// Mitsubishi GX Works2 project: PROJECT   PLC: Q03UDV

PROGRAM MAIN
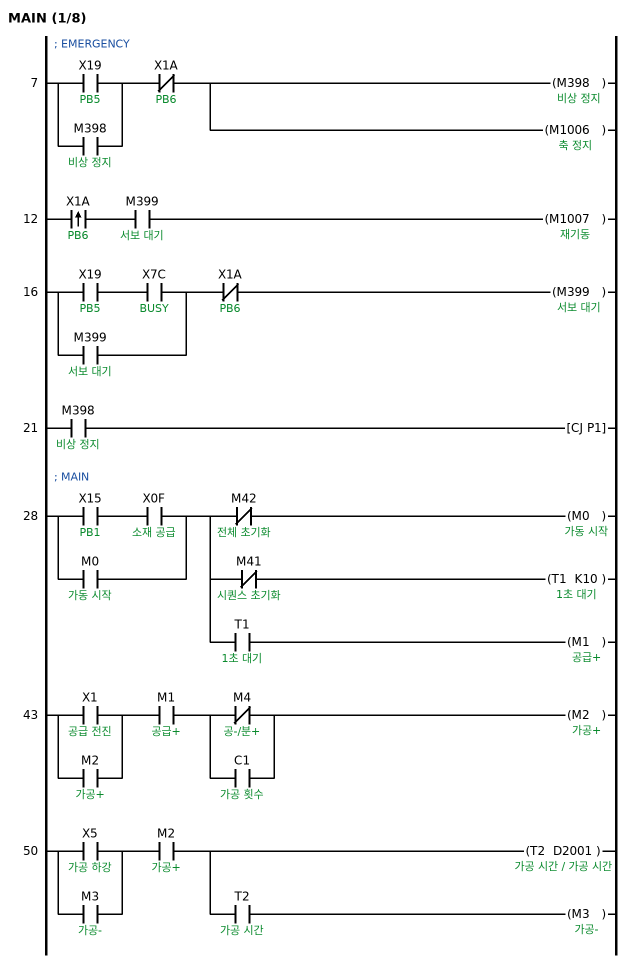
; EMERGENCY
7     LD      X19  ; PB5
      OR      M398  ; 비상 정지
      ANI     X1A  ; PB6
      OUT     M398  ; 비상 정지
      OUT     M1006  ; 축 정지
12    LDP     X1A  ; PB6
      AND     M399  ; 서보 대기
      OUT     M1007  ; 재기동
16    LD      X19  ; PB5
      AND     X7C  ; BUSY
      OR      M399  ; 서보 대기
      ANI     X1A  ; PB6
      OUT     M399  ; 서보 대기
21    LD      M398  ; 비상 정지
      CJ      P1  ; 비상 정지
; MAIN
28    LD      X15  ; PB1
      AND     X0F  ; 소재 공급
      OR      M0  ; 가동 시작
      MPS
      ANI     M42  ; 전체 초기화
      OUT     M0  ; 가동 시작
      MRD
      ANI     M41  ; 시퀀스 초기화
      OUT     T1 K10  ; 1초 대기
      MPP
      AND     T1  ; 1초 대기
      OUT     M1  ; 공급+
43    LD      X1  ; 공급 전진
      OR      M2  ; 가공+
      AND     M1  ; 공급+
      LDI     M4  ; 공-/분+
      OR      C1  ; 가공 횟수
      ANB
      OUT     M2  ; 가공+
50    LD      X5  ; 가공 하강
      OR      M3  ; 가공-
      AND     M2  ; 가공+
      OUT     T2 D2001  ; 가공 시간 / 가공 시간
      AND     T2  ; 가공 시간
      OUT     M3  ; 가공-
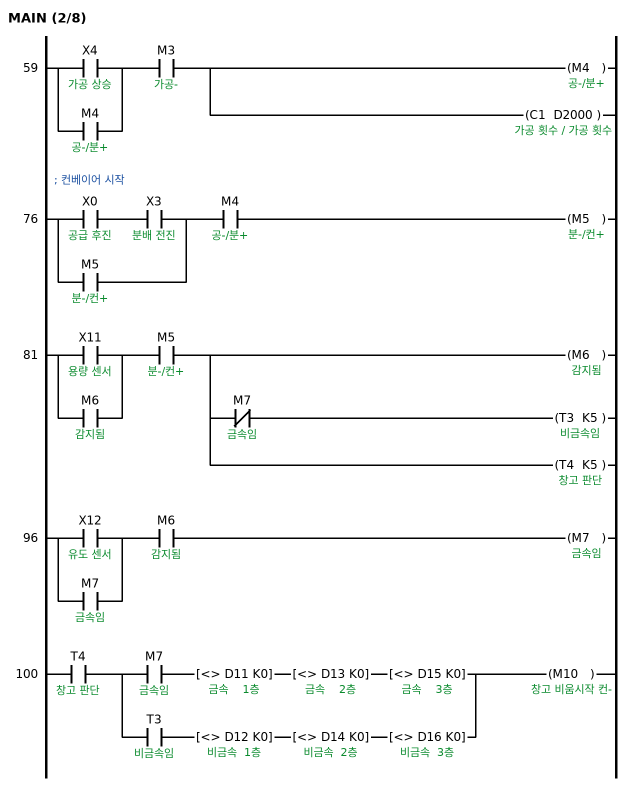
59    LD      X4  ; 가공 상승
      OR      M4  ; 공-/분+
      AND     M3  ; 가공-
      OUT     M4  ; 공-/분+
      OUT     C1 D2000  ; 가공 횟수 / 가공 횟수
; 컨베이어 시작
76    LD      X0  ; 공급 후진
      AND     X3  ; 분배 전진
      OR      M5  ; 분-/컨+
      AND     M4  ; 공-/분+
      OUT     M5  ; 분-/컨+
81    LD      X11  ; 용량 센서
      OR      M6  ; 감지됨
      AND     M5  ; 분-/컨+
      OUT     M6  ; 감지됨
      MPS
      ANI     M7  ; 금속임
      OUT     T3 K5  ; 비금속임
      MPP
      OUT     T4 K5  ; 창고 판단
96    LD      X12  ; 유도 센서
      OR      M7  ; 금속임
      AND     M6  ; 감지됨
      OUT     M7  ; 금속임
100   LD      T4  ; 창고 판단
      LD      M7  ; 금속임
      AND<>   D11 K0  ; 금속    1층
      AND<>   D13 K0  ; 금속    2층
      AND<>   D15 K0  ; 금속    3층
      LD      T3  ; 비금속임
      AND<>   D12 K0  ; 비금속  1층
      AND<>   D14 K0  ; 비금속  2층
      AND<>   D16 K0  ; 비금속  3층
      ORB
      ANB
      OUT     M10  ; 창고 비움시작 컨-
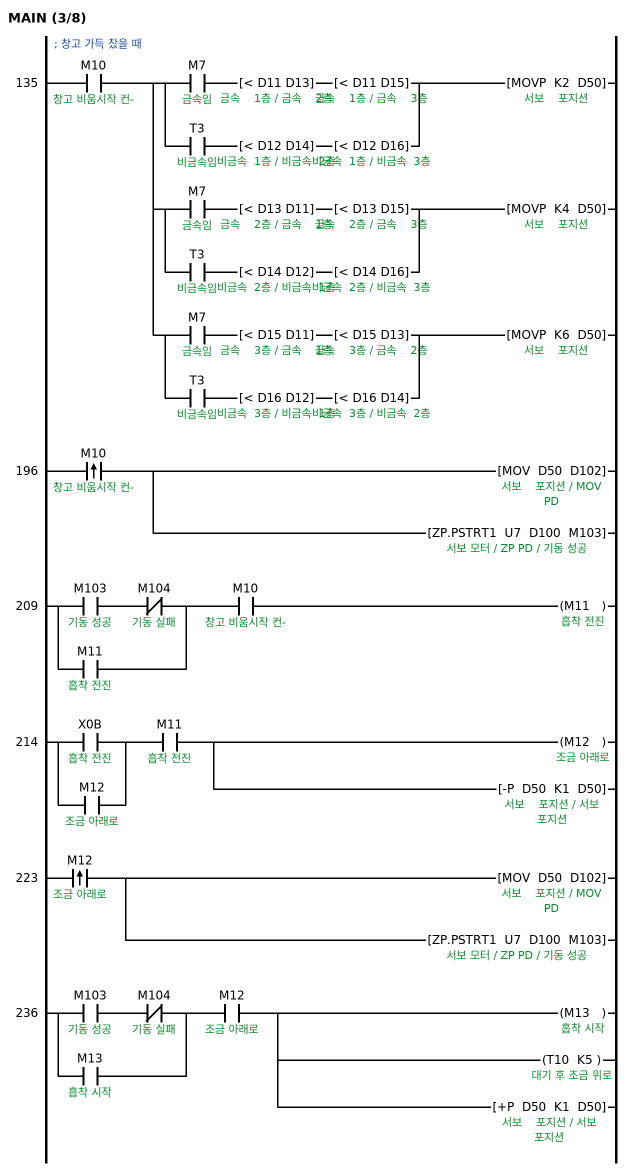
; 창고 가득 찼을 때
135   LD      M10  ; 창고 비움시작 컨-
      MPS
      LD      M7  ; 금속임
      AND<    D11 D13  ; 금속    1층 / 금속    2층
      AND<    D11 D15  ; 금속    1층 / 금속    3층
      LD      T3  ; 비금속임
      AND<    D12 D14  ; 비금속  1층 / 비금속  2층
      AND<    D12 D16  ; 비금속  1층 / 비금속  3층
      ORB
      ANB
      MOVP    K2 D50  ; 서보    포지션
      MRD
      LD      M7  ; 금속임
      AND<    D13 D11  ; 금속    2층 / 금속    1층
      AND<    D13 D15  ; 금속    2층 / 금속    3층
      LD      T3  ; 비금속임
      AND<    D14 D12  ; 비금속  2층 / 비금속  1층
      AND<    D14 D16  ; 비금속  2층 / 비금속  3층
      ORB
      ANB
      MOVP    K4 D50
      MPP
      LD      M7  ; 금속임
      AND<    D15 D11  ; 금속    3층 / 금속    1층
      AND<    D15 D13  ; 금속    3층 / 금속    2층
      LD      T3  ; 비금속임
      AND<    D16 D12  ; 비금속  3층 / 비금속  1층
      AND<    D16 D14  ; 비금속  3층 / 비금속  2층
      ORB
      ANB
      MOVP    K6 D50
196   LDP     M10  ; 창고 비움시작 컨-
      MOV     D50 D102  ; MOV PD
      ZP.PSTRT1 U7 D100 M103  ; 서보 모터 / ZP PD / 기동 성공
209   LD      M103  ; 기동 성공
      ANI     M104  ; 기동 실패
      OR      M11  ; 흡착 전진
      AND     M10  ; 창고 비움시작 컨-
      OUT     M11  ; 흡착 전진
214   LD      X0B  ; 흡착 전진
      OR      M12  ; 조금 아래로
      AND     M11  ; 흡착 전진
      OUT     M12  ; 조금 아래로
      -P      D50 K1 D50
223   LDP     M12  ; 조금 아래로
      MOV     D50 D102
      ZP.PSTRT1 U7 D100 M103
236   LD      M103  ; 기동 성공
      ANI     M104  ; 기동 실패
      OR      M13  ; 흡착 시작
      AND     M12  ; 조금 아래로
      OUT     M13  ; 흡착 시작
      OUT     T10 K5  ; 대기 후 조금 위로
      +P      D50 K1 D50
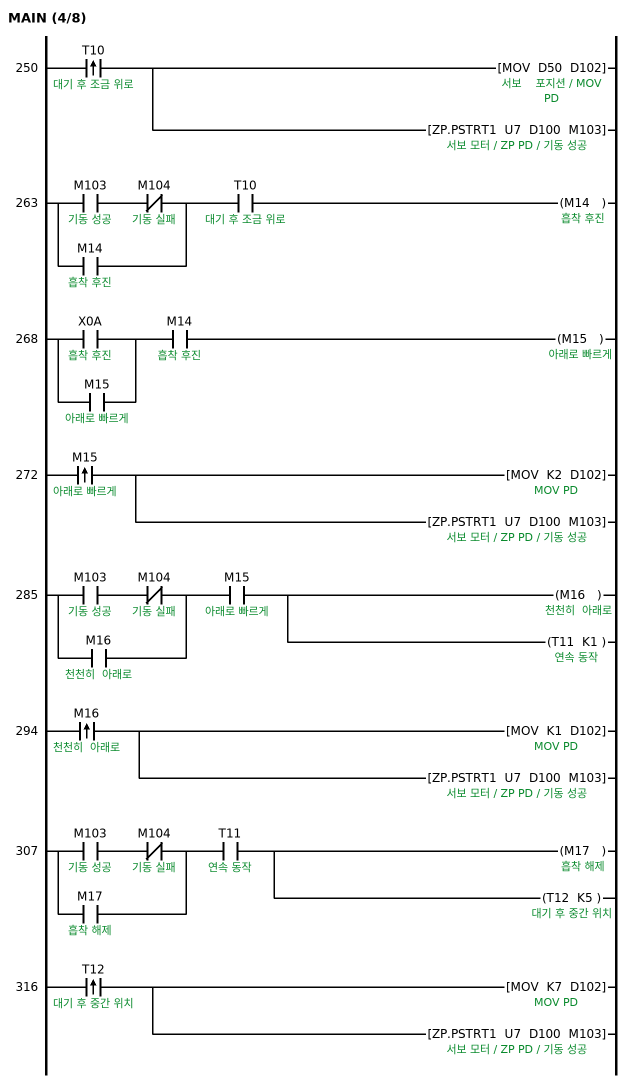
250   LDP     T10  ; 대기 후 조금 위로
      MOV     D50 D102
      ZP.PSTRT1 U7 D100 M103
263   LD      M103  ; 기동 성공
      ANI     M104  ; 기동 실패
      OR      M14  ; 흡착 후진
      AND     T10  ; 대기 후 조금 위로
      OUT     M14  ; 흡착 후진
268   LD      X0A  ; 흡착 후진
      OR      M15  ; 아래로 빠르게
      AND     M14  ; 흡착 후진
      OUT     M15  ; 아래로 빠르게
272   LDP     M15  ; 아래로 빠르게
      MOV     K2 D102
      ZP.PSTRT1 U7 D100 M103
285   LD      M103  ; 기동 성공
      ANI     M104  ; 기동 실패
      OR      M16  ; 천천히  아래로
      AND     M15  ; 아래로 빠르게
      OUT     M16  ; 천천히  아래로
      OUT     T11 K1  ; 연속 동작
294   LDP     M16  ; 천천히  아래로
      MOV     K1 D102
      ZP.PSTRT1 U7 D100 M103
307   LD      M103  ; 기동 성공
      ANI     M104  ; 기동 실패
      OR      M17  ; 흡착 해제
      AND     T11  ; 연속 동작
      OUT     M17  ; 흡착 해제
      OUT     T12 K5  ; 대기 후 중간 위치
316   LDP     T12  ; 대기 후 중간 위치
      MOV     K7 D102
      ZP.PSTRT1 U7 D100 M103
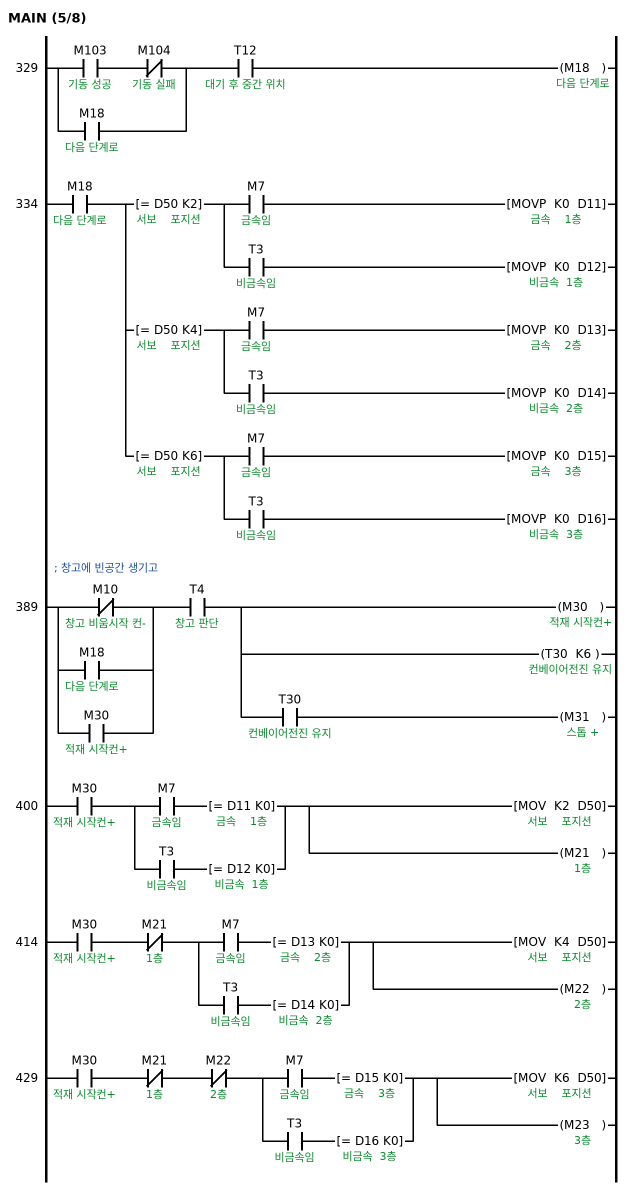
329   LD      M103  ; 기동 성공
      ANI     M104  ; 기동 실패
      OR      M18  ; 다음 단계로
      AND     T12  ; 대기 후 중간 위치
      OUT     M18  ; 다음 단계로
334   LD      M18  ; 다음 단계로
      MPS
      AND=    D50 K2  ; 서보    포지션
      MPS
      AND     M7  ; 금속임
      MOVP    K0 D11
      MPP
      AND     T3  ; 비금속임
      MOVP    K0 D12
      MRD
      AND=    D50 K4  ; 서보    포지션
      MPS
      AND     M7  ; 금속임
      MOVP    K0 D13
      MPP
      AND     T3  ; 비금속임
      MOVP    K0 D14
      MPP
      AND=    D50 K6  ; 서보    포지션
      MPS
      AND     M7  ; 금속임
      MOVP    K0 D15
      MPP
      AND     T3  ; 비금속임
      MOVP    K0 D16
; 창고에 빈공간 생기고
389   LDI     M10  ; 창고 비움시작 컨-
      OR      M18  ; 다음 단계로
      OR      M30  ; 적재 시작컨+
      AND     T4  ; 창고 판단
      OUT     M30  ; 적재 시작컨+
      OUT     T30 K6  ; 컨베이어전진 유지
      AND     T30  ; 컨베이어전진 유지
      OUT     M31  ; 스톱 +
400   LD      M30  ; 적재 시작컨+
      LD      M7  ; 금속임
      AND=    D11 K0  ; 금속    1층
      LD      T3  ; 비금속임
      AND=    D12 K0  ; 비금속  1층
      ORB
      ANB
      MOV     K2 D50
      OUT     M21  ; 1층
414   LD      M30  ; 적재 시작컨+
      ANI     M21  ; 1층
      LD      M7  ; 금속임
      AND=    D13 K0  ; 금속    2층
      LD      T3  ; 비금속임
      AND=    D14 K0  ; 비금속  2층
      ORB
      ANB
      MOV     K4 D50
      OUT     M22  ; 2층
429   LD      M30  ; 적재 시작컨+
      ANI     M21  ; 1층
      ANI     M22  ; 2층
      LD      M7  ; 금속임
      AND=    D15 K0  ; 금속    3층
      LD      T3  ; 비금속임
      AND=    D16 K0  ; 비금속  3층
      ORB
      ANB
      MOV     K6 D50
      OUT     M23  ; 3층
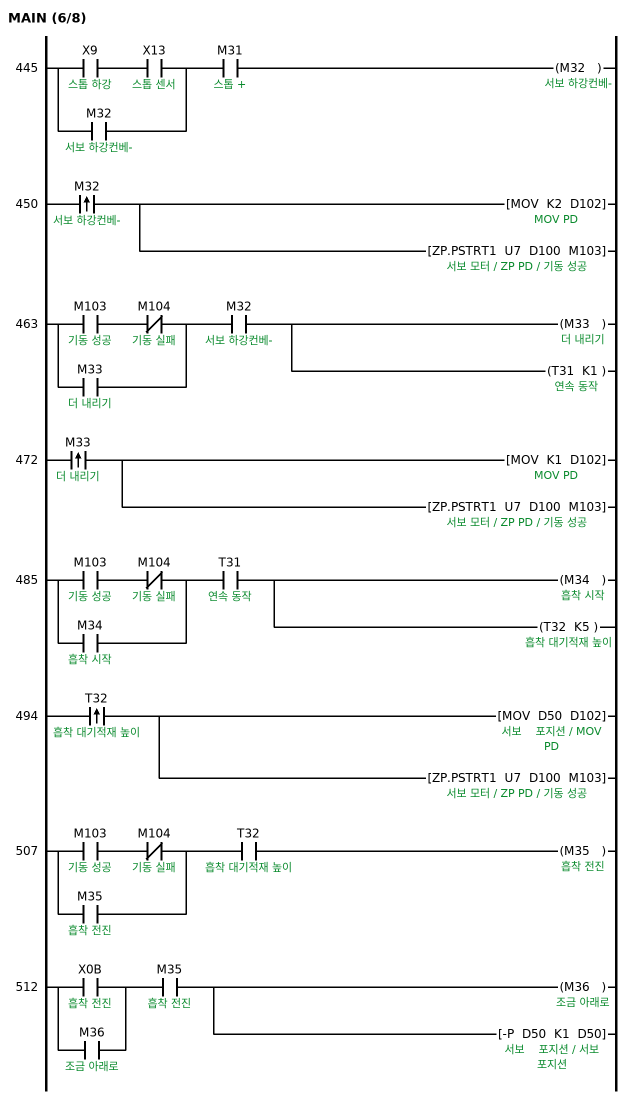
445   LD      X9  ; 스톱 하강
      AND     X13  ; 스톱 센서
      OR      M32  ; 서보 하강컨베-
      AND     M31  ; 스톱 +
      OUT     M32  ; 서보 하강컨베-
450   LDP     M32  ; 서보 하강컨베-
      MOV     K2 D102
      ZP.PSTRT1 U7 D100 M103
463   LD      M103  ; 기동 성공
      ANI     M104  ; 기동 실패
      OR      M33  ; 더 내리기
      AND     M32  ; 서보 하강컨베-
      OUT     M33  ; 더 내리기
      OUT     T31 K1  ; 연속 동작
472   LDP     M33  ; 더 내리기
      MOV     K1 D102
      ZP.PSTRT1 U7 D100 M103
485   LD      M103  ; 기동 성공
      ANI     M104  ; 기동 실패
      OR      M34  ; 흡착 시작
      AND     T31  ; 연속 동작
      OUT     M34  ; 흡착 시작
      OUT     T32 K5  ; 흡착 대기적재 높이
494   LDP     T32  ; 흡착 대기적재 높이
      MOV     D50 D102
      ZP.PSTRT1 U7 D100 M103
507   LD      M103  ; 기동 성공
      ANI     M104  ; 기동 실패
      OR      M35  ; 흡착 전진
      AND     T32  ; 흡착 대기적재 높이
      OUT     M35  ; 흡착 전진
512   LD      X0B  ; 흡착 전진
      OR      M36  ; 조금 아래로
      AND     M35  ; 흡착 전진
      OUT     M36  ; 조금 아래로
      -P      D50 K1 D50
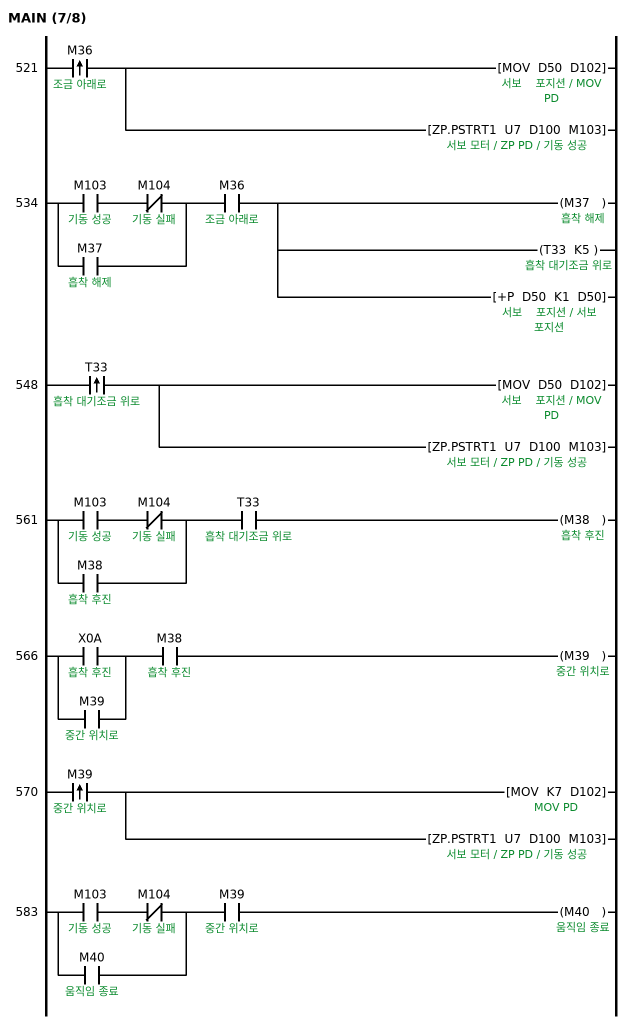
521   LDP     M36  ; 조금 아래로
      MOV     D50 D102
      ZP.PSTRT1 U7 D100 M103
534   LD      M103  ; 기동 성공
      ANI     M104  ; 기동 실패
      OR      M37  ; 흡착 해제
      AND     M36  ; 조금 아래로
      OUT     M37  ; 흡착 해제
      OUT     T33 K5  ; 흡착 대기조금 위로
      +P      D50 K1 D50
548   LDP     T33  ; 흡착 대기조금 위로
      MOV     D50 D102
      ZP.PSTRT1 U7 D100 M103
561   LD      M103  ; 기동 성공
      ANI     M104  ; 기동 실패
      OR      M38  ; 흡착 후진
      AND     T33  ; 흡착 대기조금 위로
      OUT     M38  ; 흡착 후진
566   LD      X0A  ; 흡착 후진
      OR      M39  ; 중간 위치로
      AND     M38  ; 흡착 후진
      OUT     M39  ; 중간 위치로
570   LDP     M39  ; 중간 위치로
      MOV     K7 D102
      ZP.PSTRT1 U7 D100 M103
583   LD      M103  ; 기동 성공
      ANI     M104  ; 기동 실패
      OR      M40  ; 움직임 종료
      AND     M39  ; 중간 위치로
      OUT     M40  ; 움직임 종료
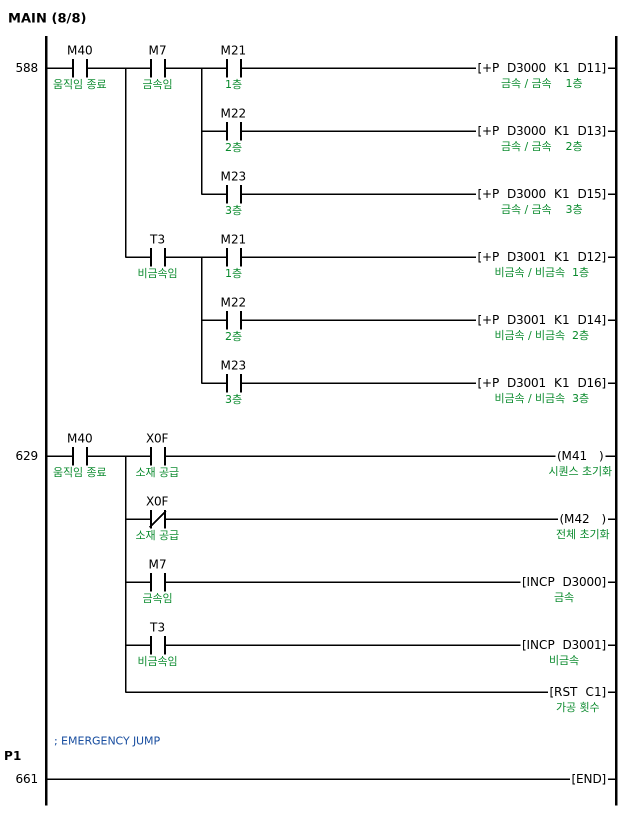
588   LD      M40  ; 움직임 종료
      MPS
      AND     M7  ; 금속임
      MPS
      AND     M21  ; 1층
      +P      D3000 K1 D11  ; 금속
      MRD
      AND     M22  ; 2층
      +P      D3000 K1 D13
      MPP
      AND     M23  ; 3층
      +P      D3000 K1 D15
      MPP
      AND     T3  ; 비금속임
      MPS
      AND     M21  ; 1층
      +P      D3001 K1 D12  ; 비금속
      MRD
      AND     M22  ; 2층
      +P      D3001 K1 D14
      MPP
      AND     M23  ; 3층
      +P      D3001 K1 D16
629   LD      M40  ; 움직임 종료
      MPS
      AND     X0F  ; 소재 공급
      OUT     M41  ; 시퀀스 초기화
      MRD
      ANI     X0F  ; 소재 공급
      OUT     M42  ; 전체 초기화
      MRD
      AND     M7  ; 금속임
      INCP    D3000
      MRD
      AND     T3  ; 비금속임
      INCP    D3001
      MPP
      RST     C1  ; 가공 횟수
; EMERGENCY JUMP
      P1
661   END
END_PROGRAM

PROGRAM INIT
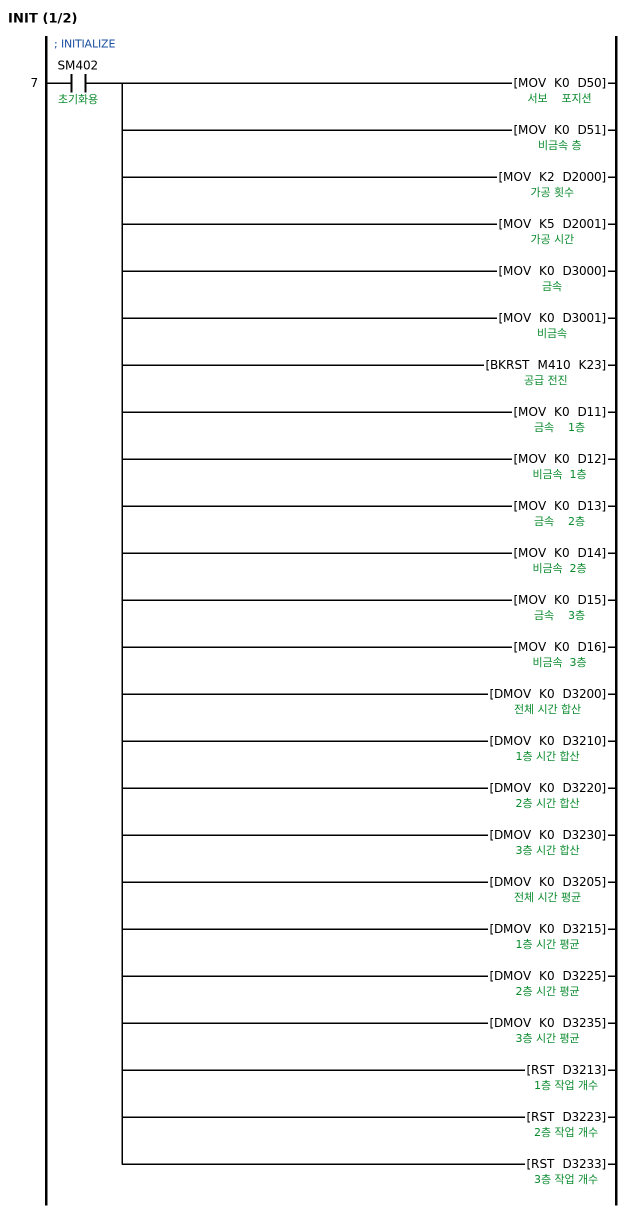
; INITIALIZE
7     LD      SM402  ; 초기화용
      MOV     K0 D50  ; 서보    포지션
      MOV     K0 D51  ; 비금속 층
      MOV     K2 D2000  ; 가공 횟수
      MOV     K5 D2001  ; 가공 시간
      MOV     K0 D3000  ; 금속
      MOV     K0 D3001  ; 비금속
      BKRST   M410 K23  ; 공급 전진
      MOV     K0 D11  ; 금속    1층
      MOV     K0 D12  ; 비금속  1층
      MOV     K0 D13  ; 금속    2층
      MOV     K0 D14  ; 비금속  2층
      MOV     K0 D15  ; 금속    3층
      MOV     K0 D16  ; 비금속  3층
      DMOV    K0 D3200  ; 전체 시간 합산
      DMOV    K0 D3210  ; 1층 시간 합산
      DMOV    K0 D3220  ; 2층 시간 합산
      DMOV    K0 D3230  ; 3층 시간 합산
      DMOV    K0 D3205  ; 전체 시간 평균
      DMOV    K0 D3215  ; 1층 시간 평균
      DMOV    K0 D3225  ; 2층 시간 평균
      DMOV    K0 D3235  ; 3층 시간 평균
      RST     D3213  ; 1층 작업 개수
      RST     D3223  ; 2층 작업 개수
      RST     D3233  ; 3층 작업 개수
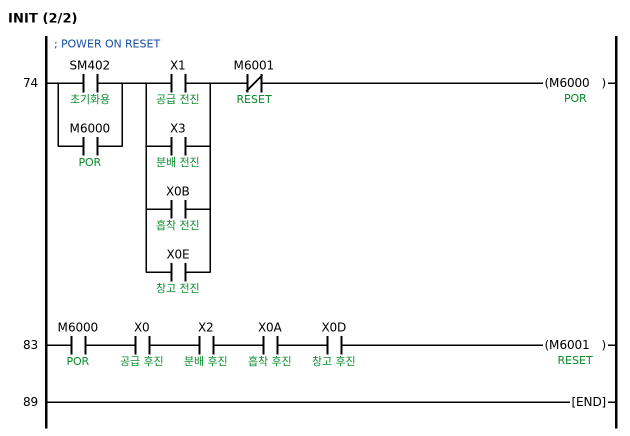
; POWER ON RESET
74    LD      SM402  ; 초기화용
      OR      M6000  ; POR
      LD      X1  ; 공급 전진
      OR      X3  ; 분배 전진
      OR      X0B  ; 흡착 전진
      OR      X0E  ; 창고 전진
      ANB
      ANI     M6001  ; RESET
      OUT     M6000  ; POR
83    LD      M6000  ; POR
      AND     X0  ; 공급 후진
      AND     X2  ; 분배 후진
      AND     X0A  ; 흡착 후진
      AND     X0D  ; 창고 후진
      OUT     M6001  ; RESET
89    END
END_PROGRAM

PROGRAM UNLOAD2
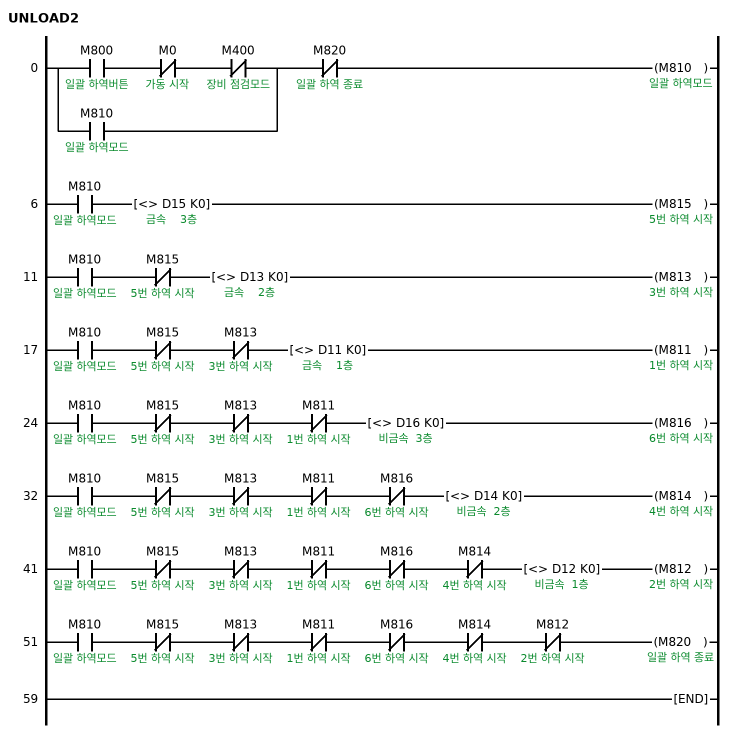
0     LD      M800  ; 일괄 하역버튼
      ANI     M0  ; 가동 시작
      ANI     M400  ; 장비 점검모드
      OR      M810  ; 일괄 하역모드
      ANI     M820  ; 일괄 하역 종료
      OUT     M810  ; 일괄 하역모드
6     LD      M810  ; 일괄 하역모드
      AND<>   D15 K0  ; 금속    3층
      OUT     M815  ; 5번 하역 시작
11    LD      M810  ; 일괄 하역모드
      ANI     M815  ; 5번 하역 시작
      AND<>   D13 K0  ; 금속    2층
      OUT     M813  ; 3번 하역 시작
17    LD      M810  ; 일괄 하역모드
      ANI     M815  ; 5번 하역 시작
      ANI     M813  ; 3번 하역 시작
      AND<>   D11 K0  ; 금속    1층
      OUT     M811  ; 1번 하역 시작
24    LD      M810  ; 일괄 하역모드
      ANI     M815  ; 5번 하역 시작
      ANI     M813  ; 3번 하역 시작
      ANI     M811  ; 1번 하역 시작
      AND<>   D16 K0  ; 비금속  3층
      OUT     M816  ; 6번 하역 시작
32    LD      M810  ; 일괄 하역모드
      ANI     M815  ; 5번 하역 시작
      ANI     M813  ; 3번 하역 시작
      ANI     M811  ; 1번 하역 시작
      ANI     M816  ; 6번 하역 시작
      AND<>   D14 K0  ; 비금속  2층
      OUT     M814  ; 4번 하역 시작
41    LD      M810  ; 일괄 하역모드
      ANI     M815  ; 5번 하역 시작
      ANI     M813  ; 3번 하역 시작
      ANI     M811  ; 1번 하역 시작
      ANI     M816  ; 6번 하역 시작
      ANI     M814  ; 4번 하역 시작
      AND<>   D12 K0  ; 비금속  1층
      OUT     M812  ; 2번 하역 시작
51    LD      M810  ; 일괄 하역모드
      ANI     M815  ; 5번 하역 시작
      ANI     M813  ; 3번 하역 시작
      ANI     M811  ; 1번 하역 시작
      ANI     M816  ; 6번 하역 시작
      ANI     M814  ; 4번 하역 시작
      ANI     M812  ; 2번 하역 시작
      OUT     M820  ; 일괄 하역 종료
59    END
END_PROGRAM

PROGRAM TEST
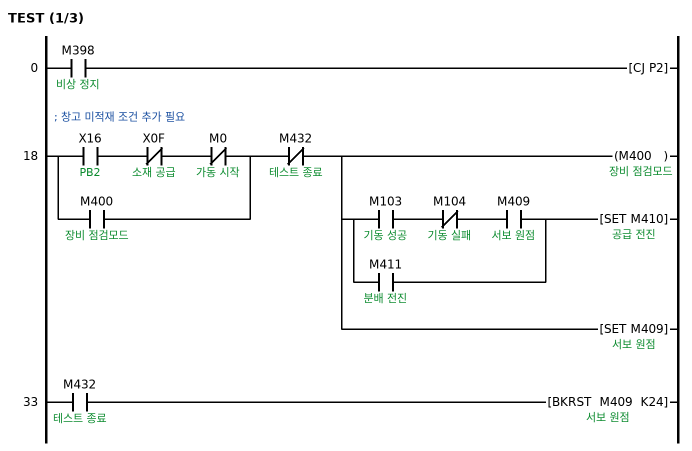
0     LD      M398  ; 비상 정지
      CJ      P2  ; 비상 정지
; 창고 미적재 조건 추가 필요
18    LD      X16  ; PB2
      ANI     X0F  ; 소재 공급
      ANI     M0  ; 가동 시작
      OR      M400  ; 장비 점검모드
      ANI     M432  ; 테스트 종료
      OUT     M400  ; 장비 점검모드
      MPS
      LD      M103  ; 기동 성공
      ANI     M104  ; 기동 실패
      AND     M409  ; 서보 원점
      OR      M411  ; 분배 전진
      ANB
      SET     M410  ; 공급 전진
      MPP
      SET     M409  ; 서보 원점
33    LD      M432  ; 테스트 종료
      BKRST   M409 K24
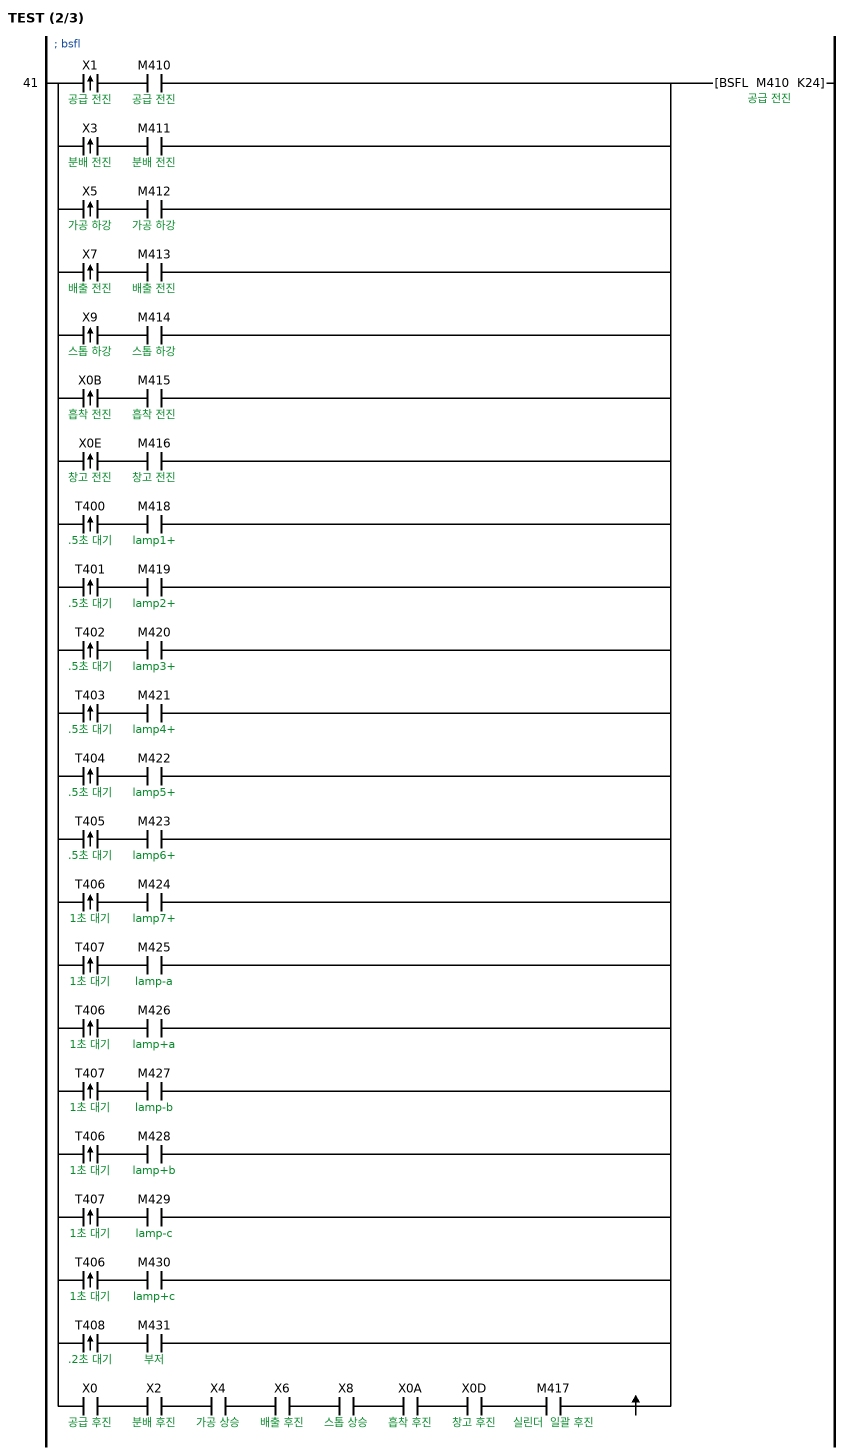
; bsfl
41    LDP     X1  ; 공급 전진
      AND     M410  ; 공급 전진
      LDP     X3  ; 분배 전진
      AND     M411  ; 분배 전진
      ORB
      LDP     X5  ; 가공 하강
      AND     M412  ; 가공 하강
      ORB
      LDP     X7  ; 배출 전진
      AND     M413  ; 배출 전진
      ORB
      LDP     X9  ; 스톱 하강
      AND     M414  ; 스톱 하강
      ORB
      LDP     X0B  ; 흡착 전진
      AND     M415  ; 흡착 전진
      ORB
      LDP     X0E  ; 창고 전진
      AND     M416  ; 창고 전진
      ORB
      LDP     T400  ; .5초 대기
      AND     M418  ; lamp1+
      ORB
      LDP     T401  ; .5초 대기
      AND     M419  ; lamp2+
      ORB
      LDP     T402  ; .5초 대기
      AND     M420  ; lamp3+
      ORB
      LDP     T403  ; .5초 대기
      AND     M421  ; lamp4+
      ORB
      LDP     T404  ; .5초 대기
      AND     M422  ; lamp5+
      ORB
      LDP     T405  ; .5초 대기
      AND     M423  ; lamp6+
      ORB
      LDP     T406  ; 1초 대기
      AND     M424  ; lamp7+
      ORB
      LDP     T407  ; 1초 대기
      AND     M425  ; lamp-a
      ORB
      LDP     T406  ; 1초 대기
      AND     M426  ; lamp+a
      ORB
      LDP     T407  ; 1초 대기
      AND     M427  ; lamp-b
      ORB
      LDP     T406  ; 1초 대기
      AND     M428  ; lamp+b
      ORB
      LDP     T407  ; 1초 대기
      AND     M429  ; lamp-c
      ORB
      LDP     T406  ; 1초 대기
      AND     M430  ; lamp+c
      ORB
      LDP     T408  ; .2초 대기
      AND     M431  ; 부저
      ORB
      LD      X0  ; 공급 후진
      AND     X2  ; 분배 후진
      AND     X4  ; 가공 상승
      AND     X6  ; 배출 후진
      AND     X8  ; 스톱 상승
      AND     X0A  ; 흡착 후진
      AND     X0D  ; 창고 후진
      AND     M417  ; 실린더  일괄 후진
      MEP
      ORB
      BSFL    M410 K24
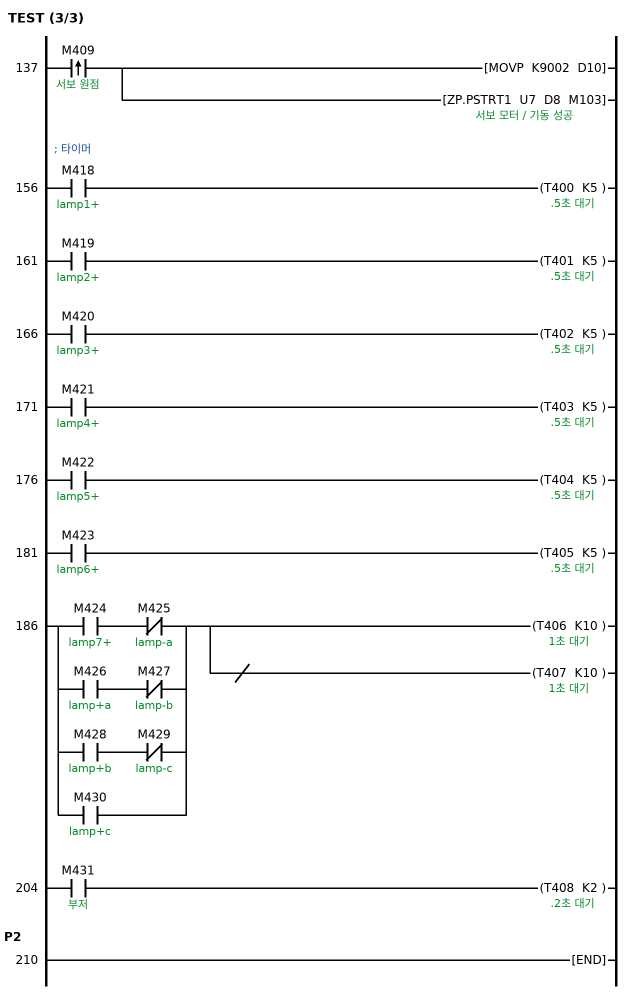
137   LDP     M409  ; 서보 원점
      MOVP    K9002 D10
      ZP.PSTRT1 U7 D8 M103  ; 서보 모터
; 타이머
156   LD      M418  ; lamp1+
      OUT     T400 K5  ; .5초 대기
161   LD      M419  ; lamp2+
      OUT     T401 K5  ; .5초 대기
166   LD      M420  ; lamp3+
      OUT     T402 K5  ; .5초 대기
171   LD      M421  ; lamp4+
      OUT     T403 K5  ; .5초 대기
176   LD      M422  ; lamp5+
      OUT     T404 K5  ; .5초 대기
181   LD      M423  ; lamp6+
      OUT     T405 K5  ; .5초 대기
186   LD      M424  ; lamp7+
      ANI     M425  ; lamp-a
      LD      M426  ; lamp+a
      ANI     M427  ; lamp-b
      ORB
      LD      M428  ; lamp+b
      ANI     M429  ; lamp-c
      ORB
      OR      M430  ; lamp+c
      OUT     T406 K10  ; 1초 대기
      INV
      OUT     T407 K10  ; 1초 대기
204   LD      M431  ; 부저
      OUT     T408 K2  ; .2초 대기
      P2
210   END
END_PROGRAM

PROGRAM OUTPUT
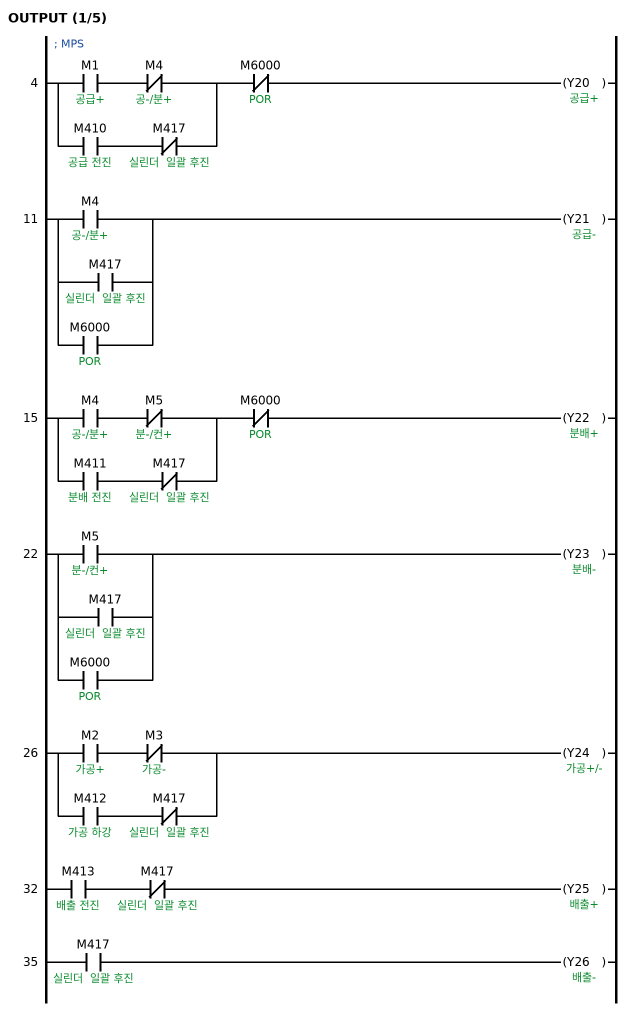
; MPS
4     LD      M1  ; 공급+
      ANI     M4  ; 공-/분+
      LD      M410  ; 공급 전진
      ANI     M417  ; 실린더  일괄 후진
      ORB
      ANI     M6000  ; POR
      OUT     Y20  ; 공급+
11    LD      M4  ; 공-/분+
      OR      M417  ; 실린더  일괄 후진
      OR      M6000  ; POR
      OUT     Y21  ; 공급-
15    LD      M4  ; 공-/분+
      ANI     M5  ; 분-/컨+
      LD      M411  ; 분배 전진
      ANI     M417  ; 실린더  일괄 후진
      ORB
      ANI     M6000  ; POR
      OUT     Y22  ; 분배+
22    LD      M5  ; 분-/컨+
      OR      M417  ; 실린더  일괄 후진
      OR      M6000  ; POR
      OUT     Y23  ; 분배-
26    LD      M2  ; 가공+
      ANI     M3  ; 가공-
      LD      M412  ; 가공 하강
      ANI     M417  ; 실린더  일괄 후진
      ORB
      OUT     Y24  ; 가공+/-
32    LD      M413  ; 배출 전진
      ANI     M417  ; 실린더  일괄 후진
      OUT     Y25  ; 배출+
35    LD      M417  ; 실린더  일괄 후진
      OUT     Y26  ; 배출-
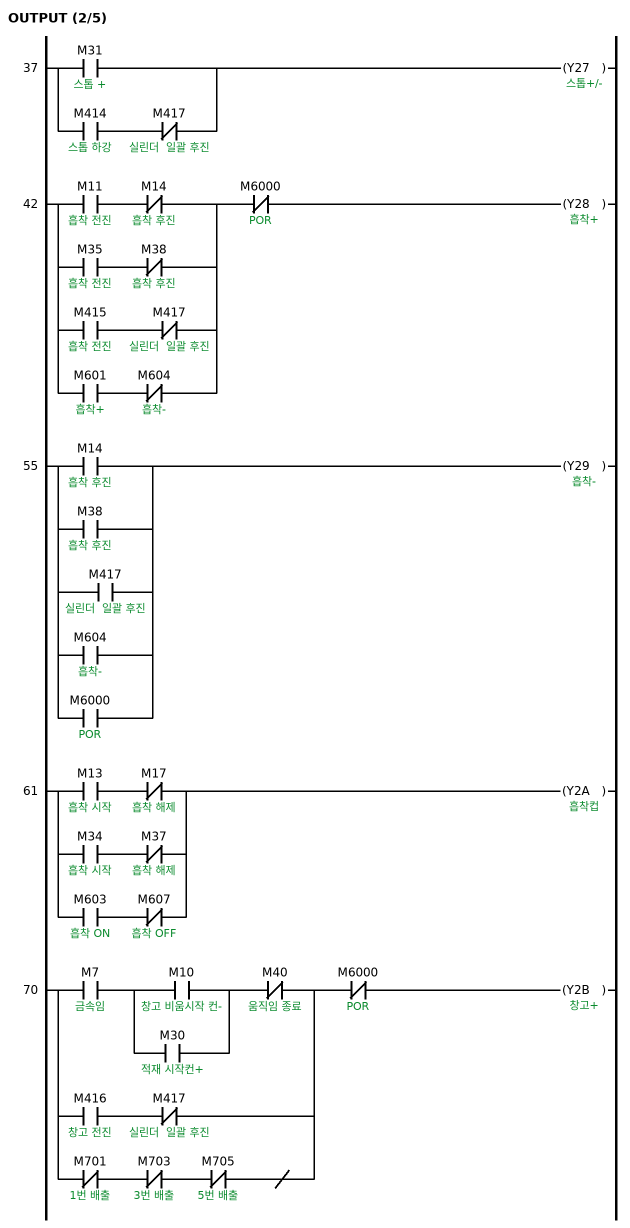
37    LD      M31  ; 스톱 +
      LD      M414  ; 스톱 하강
      ANI     M417  ; 실린더  일괄 후진
      ORB
      OUT     Y27  ; 스톱+/-
42    LD      M11  ; 흡착 전진
      ANI     M14  ; 흡착 후진
      LD      M35  ; 흡착 전진
      ANI     M38  ; 흡착 후진
      ORB
      LD      M415  ; 흡착 전진
      ANI     M417  ; 실린더  일괄 후진
      ORB
      LD      M601  ; 흡착+
      ANI     M604  ; 흡착-
      ORB
      ANI     M6000  ; POR
      OUT     Y28  ; 흡착+
55    LD      M14  ; 흡착 후진
      OR      M38  ; 흡착 후진
      OR      M417  ; 실린더  일괄 후진
      OR      M604  ; 흡착-
      OR      M6000  ; POR
      OUT     Y29  ; 흡착-
61    LD      M13  ; 흡착 시작
      ANI     M17  ; 흡착 해제
      LD      M34  ; 흡착 시작
      ANI     M37  ; 흡착 해제
      ORB
      LD      M603  ; 흡착 ON
      ANI     M607  ; 흡착 OFF
      ORB
      OUT     Y2A  ; 흡착컵
70    LD      M7  ; 금속임
      LD      M10  ; 창고 비움시작 컨-
      OR      M30  ; 적재 시작컨+
      ANB
      ANI     M40  ; 움직임 종료
      LD      M416  ; 창고 전진
      ANI     M417  ; 실린더  일괄 후진
      ORB
      LDI     M701  ; 1번 배출
      ANI     M703  ; 3번 배출
      ANI     M705  ; 5번 배출
      INV
      ORB
      ANI     M6000  ; POR
      OUT     Y2B  ; 창고+
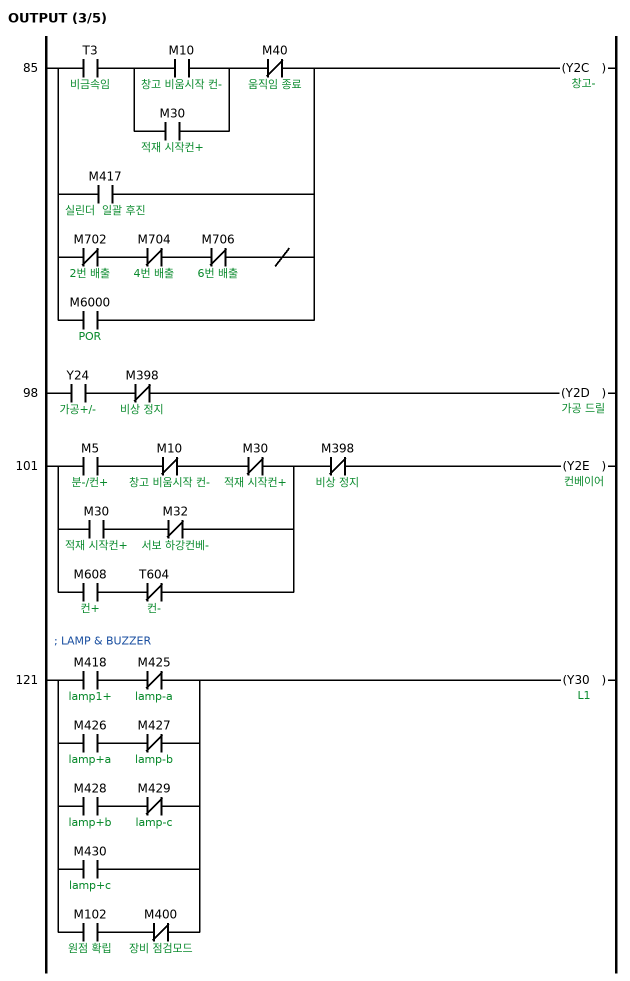
85    LD      T3  ; 비금속임
      LD      M10  ; 창고 비움시작 컨-
      OR      M30  ; 적재 시작컨+
      ANB
      ANI     M40  ; 움직임 종료
      OR      M417  ; 실린더  일괄 후진
      LDI     M702  ; 2번 배출
      ANI     M704  ; 4번 배출
      ANI     M706  ; 6번 배출
      INV
      ORB
      OR      M6000  ; POR
      OUT     Y2C  ; 창고-
98    LD      Y24  ; 가공+/-
      ANI     M398  ; 비상 정지
      OUT     Y2D  ; 가공 드릴
101   LD      M5  ; 분-/컨+
      ANI     M10  ; 창고 비움시작 컨-
      ANI     M30  ; 적재 시작컨+
      LD      M30  ; 적재 시작컨+
      ANI     M32  ; 서보 하강컨베-
      ORB
      LD      M608  ; 컨+
      ANI     T604  ; 컨-
      ORB
      ANI     M398  ; 비상 정지
      OUT     Y2E  ; 컨베이어
; LAMP & BUZZER
121   LD      M418  ; lamp1+
      ANI     M425  ; lamp-a
      LD      M426  ; lamp+a
      ANI     M427  ; lamp-b
      ORB
      LD      M428  ; lamp+b
      ANI     M429  ; lamp-c
      ORB
      OR      M430  ; lamp+c
      LD      M102  ; 원점 확립
      ANI     M400  ; 장비 점검모드
      ORB
      OUT     Y30  ; L1
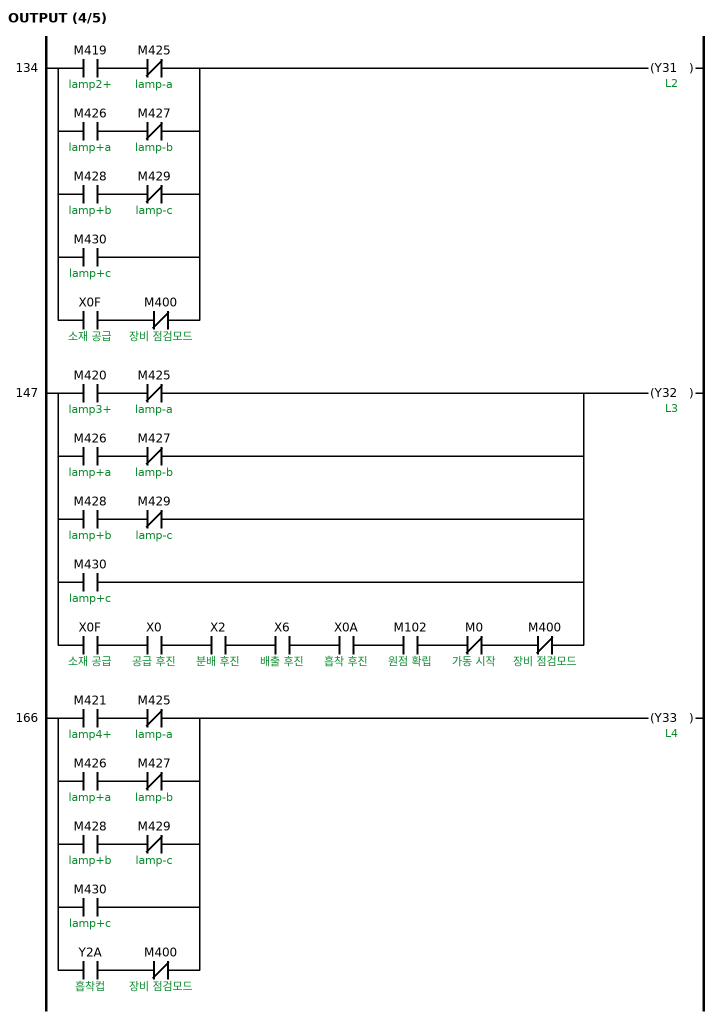
134   LD      M419  ; lamp2+
      ANI     M425  ; lamp-a
      LD      M426  ; lamp+a
      ANI     M427  ; lamp-b
      ORB
      LD      M428  ; lamp+b
      ANI     M429  ; lamp-c
      ORB
      OR      M430  ; lamp+c
      LD      X0F  ; 소재 공급
      ANI     M400  ; 장비 점검모드
      ORB
      OUT     Y31  ; L2
147   LD      M420  ; lamp3+
      ANI     M425  ; lamp-a
      LD      M426  ; lamp+a
      ANI     M427  ; lamp-b
      ORB
      LD      M428  ; lamp+b
      ANI     M429  ; lamp-c
      ORB
      OR      M430  ; lamp+c
      LD      X0F  ; 소재 공급
      AND     X0  ; 공급 후진
      AND     X2  ; 분배 후진
      AND     X6  ; 배출 후진
      AND     X0A  ; 흡착 후진
      AND     M102  ; 원점 확립
      ANI     M0  ; 가동 시작
      ANI     M400  ; 장비 점검모드
      ORB
      OUT     Y32  ; L3
166   LD      M421  ; lamp4+
      ANI     M425  ; lamp-a
      LD      M426  ; lamp+a
      ANI     M427  ; lamp-b
      ORB
      LD      M428  ; lamp+b
      ANI     M429  ; lamp-c
      ORB
      OR      M430  ; lamp+c
      LD      Y2A  ; 흡착컵
      ANI     M400  ; 장비 점검모드
      ORB
      OUT     Y33  ; L4
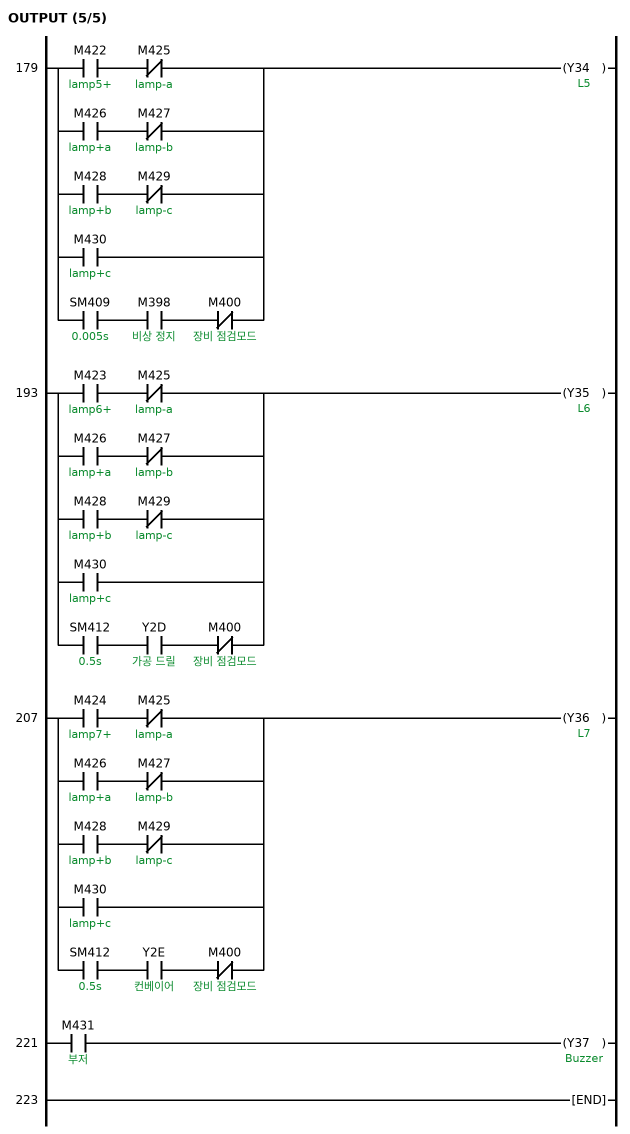
179   LD      M422  ; lamp5+
      ANI     M425  ; lamp-a
      LD      M426  ; lamp+a
      ANI     M427  ; lamp-b
      ORB
      LD      M428  ; lamp+b
      ANI     M429  ; lamp-c
      ORB
      OR      M430  ; lamp+c
      LD      SM409  ; 0.005s
      AND     M398  ; 비상 정지
      ANI     M400  ; 장비 점검모드
      ORB
      OUT     Y34  ; L5
193   LD      M423  ; lamp6+
      ANI     M425  ; lamp-a
      LD      M426  ; lamp+a
      ANI     M427  ; lamp-b
      ORB
      LD      M428  ; lamp+b
      ANI     M429  ; lamp-c
      ORB
      OR      M430  ; lamp+c
      LD      SM412  ; 0.5s
      AND     Y2D  ; 가공 드릴
      ANI     M400  ; 장비 점검모드
      ORB
      OUT     Y35  ; L6
207   LD      M424  ; lamp7+
      ANI     M425  ; lamp-a
      LD      M426  ; lamp+a
      ANI     M427  ; lamp-b
      ORB
      LD      M428  ; lamp+b
      ANI     M429  ; lamp-c
      ORB
      OR      M430  ; lamp+c
      LD      SM412  ; 0.5s
      AND     Y2E  ; 컨베이어
      ANI     M400  ; 장비 점검모드
      ORB
      OUT     Y36  ; L7
221   LD      M431  ; 부저
      OUT     Y37  ; Buzzer
223   END
END_PROGRAM

PROGRAM STAT
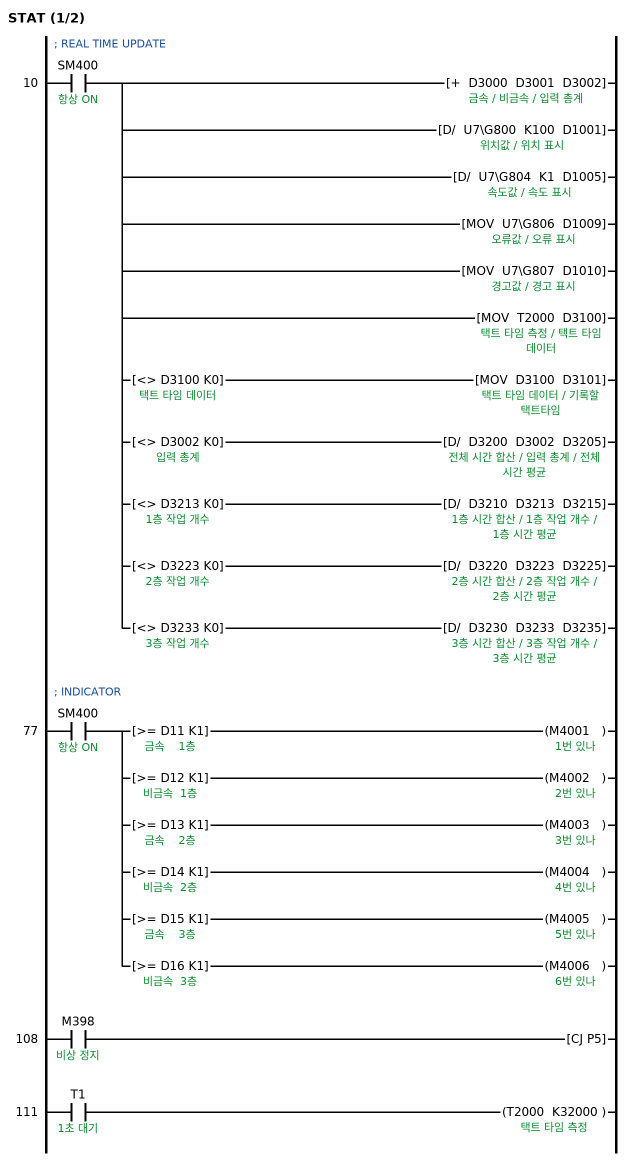
; REAL TIME UPDATE
10    LD      SM400  ; 항상 ON
      +       D3000 D3001 D3002  ; 금속 / 비금속 / 입력 총계
      D/      U7\G800 K100 D1001  ; 위치값 / 위치 표시
      D/      U7\G804 K1 D1005  ; 속도값 / 속도 표시
      MOV     U7\G806 D1009  ; 오류값 / 오류 표시
      MOV     U7\G807 D1010  ; 경고값 / 경고 표시
      MOV     T2000 D3100  ; 택트 타임 측정 / 택트 타임 데이터
      MPS
      AND<>   D3100 K0  ; 택트 타임 데이터
      MOV     D3100 D3101  ; 기록할  택트타임
      MRD
      AND<>   D3002 K0  ; 입력 총계
      D/      D3200 D3002 D3205  ; 전체 시간 합산 / 전체 시간 평균
      MRD
      AND<>   D3213 K0  ; 1층 작업 개수
      D/      D3210 D3213 D3215  ; 1층 시간 합산 / 1층 시간 평균
      MRD
      AND<>   D3223 K0  ; 2층 작업 개수
      D/      D3220 D3223 D3225  ; 2층 시간 합산 / 2층 시간 평균
      MPP
      AND<>   D3233 K0  ; 3층 작업 개수
      D/      D3230 D3233 D3235  ; 3층 시간 합산 / 3층 시간 평균
; INDICATOR
77    LD      SM400  ; 항상 ON
      MPS
      AND>=   D11 K1  ; 금속    1층
      OUT     M4001  ; 1번 있나
      MRD
      AND>=   D12 K1  ; 비금속  1층
      OUT     M4002  ; 2번 있나
      MRD
      AND>=   D13 K1  ; 금속    2층
      OUT     M4003  ; 3번 있나
      MRD
      AND>=   D14 K1  ; 비금속  2층
      OUT     M4004  ; 4번 있나
      MRD
      AND>=   D15 K1  ; 금속    3층
      OUT     M4005  ; 5번 있나
      MPP
      AND>=   D16 K1  ; 비금속  3층
      OUT     M4006  ; 6번 있나
108   LD      M398  ; 비상 정지
      CJ      P5  ; 비상정지
111   LD      T1  ; 1초 대기
      OUT     T2000 K32000  ; 택트 타임 측정
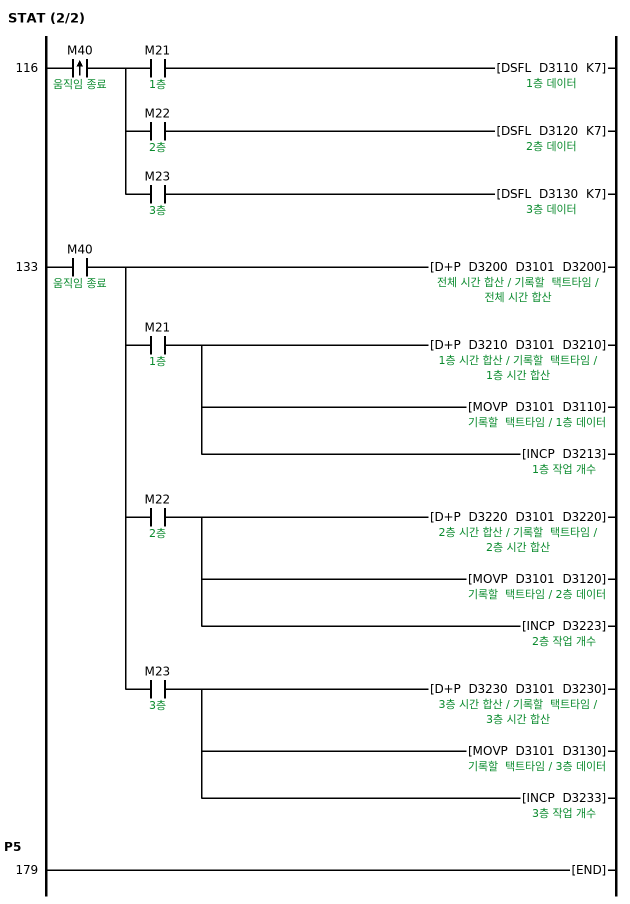
116   LDP     M40  ; 움직임 종료
      MPS
      AND     M21  ; 1층
      DSFL    D3110 K7  ; 1층 데이터
      MRD
      AND     M22  ; 2층
      DSFL    D3120 K7  ; 2층 데이터
      MPP
      AND     M23  ; 3층
      DSFL    D3130 K7  ; 3층 데이터
133   LD      M40  ; 움직임 종료
      D+P     D3200 D3101 D3200
      MPS
      AND     M21  ; 1층
      D+P     D3210 D3101 D3210
      MOVP    D3101 D3110
      INCP    D3213
      MRD
      AND     M22  ; 2층
      D+P     D3220 D3101 D3220
      MOVP    D3101 D3120
      INCP    D3223
      MPP
      AND     M23  ; 3층
      D+P     D3230 D3101 D3230
      MOVP    D3101 D3130
      INCP    D3233
      P5
179   END
END_PROGRAM

PROGRAM SERVO
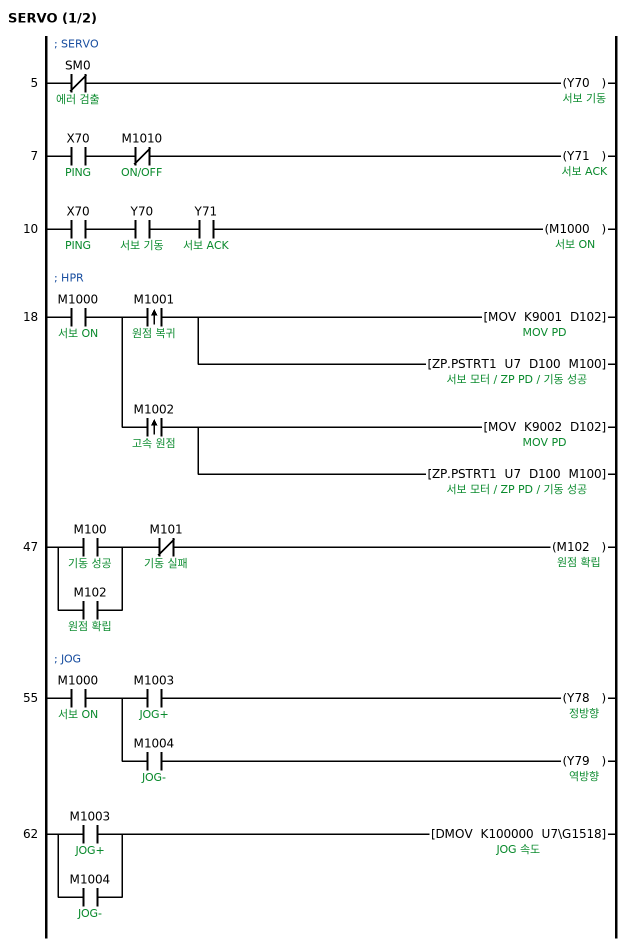
; SERVO
5     LDI     SM0  ; 에러 검출
      OUT     Y70  ; 서보 기동
7     LD      X70  ; PING
      ANI     M1010  ; ON/OFF
      OUT     Y71  ; 서보 ACK
10    LD      X70  ; PING
      AND     Y70  ; 서보 기동
      AND     Y71  ; 서보 ACK
      OUT     M1000  ; 서보 ON
; HPR
18    LD      M1000  ; 서보 ON
      MPS
      ANDP    M1001  ; 원점 복귀
      MOV     K9001 D102  ; MOV PD
      ZP.PSTRT1 U7 D100 M100  ; 서보 모터 / ZP PD / 기동 성공
      MPP
      ANDP    M1002  ; 고속 원점
      MOV     K9002 D102
      ZP.PSTRT1 U7 D100 M100
47    LD      M100  ; 기동 성공
      OR      M102  ; 원점 확립
      ANI     M101  ; 기동 실패
      OUT     M102  ; 원점 확립
; JOG
55    LD      M1000  ; 서보 ON
      MPS
      AND     M1003  ; JOG+
      OUT     Y78  ; 정방향
      MPP
      AND     M1004  ; JOG-
      OUT     Y79  ; 역방향
62    LD      M1003  ; JOG+
      OR      M1004  ; JOG-
      DMOV    K100000 U7\G1518  ; JOG 속도
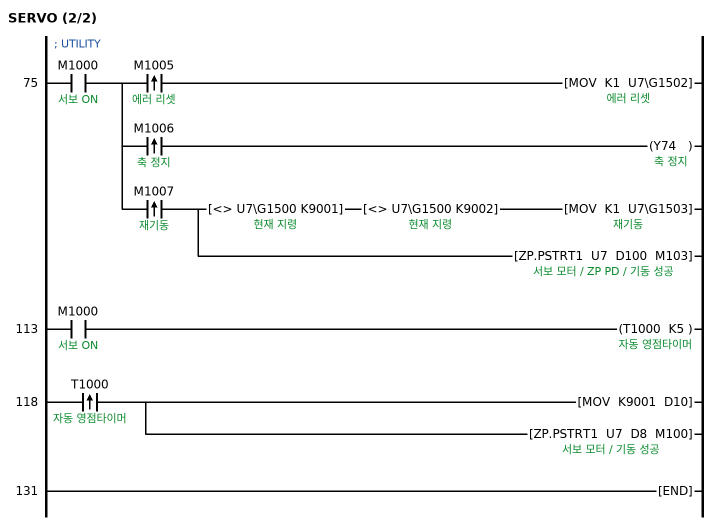
; UTILITY
75    LD      M1000  ; 서보 ON
      MPS
      ANDP    M1005  ; 에러 리셋
      MOV     K1 U7\G1502  ; 에러 리셋
      MRD
      ANDP    M1006  ; 축 정지
      OUT     Y74  ; 축 정지
      MPP
      ANDP    M1007  ; 재기동
      MPS
      AND<>   U7\G1500 K9001  ; 현재 지령
      AND<>   U7\G1500 K9002  ; 현재 지령
      MOV     K1 U7\G1503  ; 재기동
      MPP
      ZP.PSTRT1 U7 D100 M103  ; 기동 성공
113   LD      M1000  ; 서보 ON
      OUT     T1000 K5  ; 자동 영점타이머
118   LDP     T1000  ; 자동 영점타이머
      MOV     K9001 D10
      ZP.PSTRT1 U7 D8 M100
131   END
END_PROGRAM

PROGRAM UNLOAD1
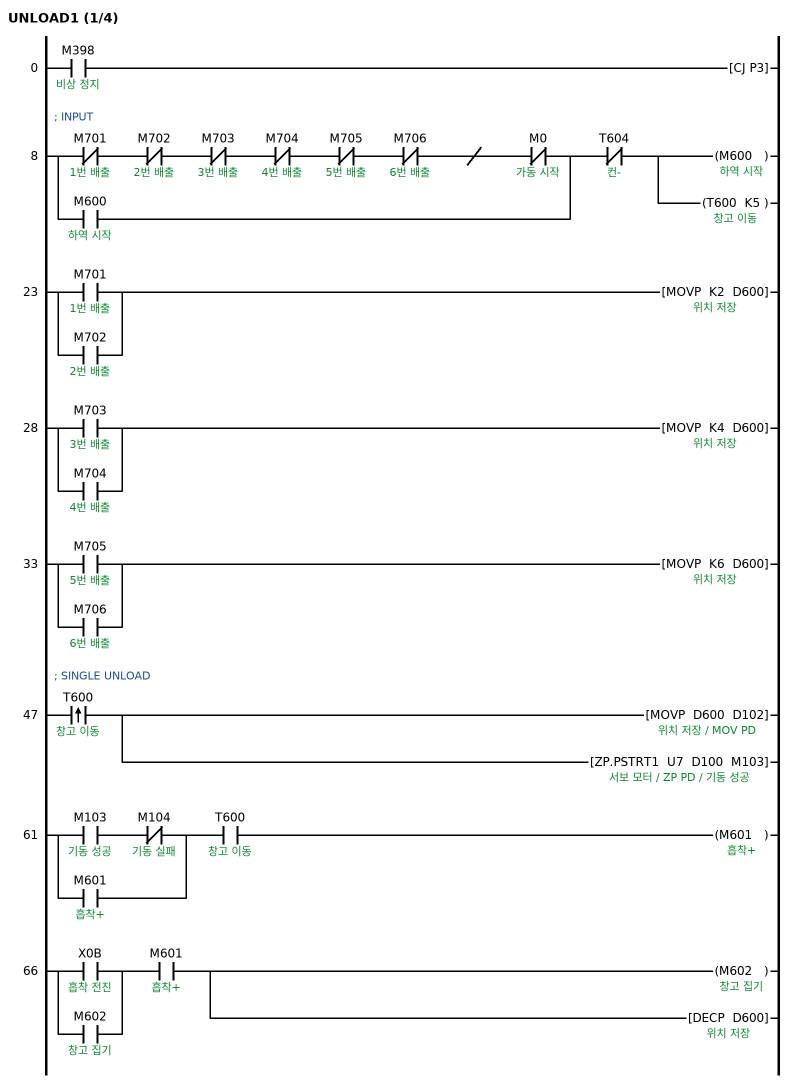
0     LD      M398  ; 비상 정지
      CJ      P3  ; 비상정지
; INPUT
8     LDI     M701  ; 1번 배출
      ANI     M702  ; 2번 배출
      ANI     M703  ; 3번 배출
      ANI     M704  ; 4번 배출
      ANI     M705  ; 5번 배출
      ANI     M706  ; 6번 배출
      INV
      ANI     M0  ; 가동 시작
      OR      M600  ; 하역 시작
      ANI     T604  ; 컨-
      OUT     M600  ; 하역 시작
      OUT     T600 K5  ; 창고 이동
23    LD      M701  ; 1번 배출
      OR      M702  ; 2번 배출
      MOVP    K2 D600  ; 위치 저장
28    LD      M703  ; 3번 배출
      OR      M704  ; 4번 배출
      MOVP    K4 D600
33    LD      M705  ; 5번 배출
      OR      M706  ; 6번 배출
      MOVP    K6 D600
; SINGLE UNLOAD
47    LDP     T600  ; 창고 이동
      MOVP    D600 D102  ; MOV PD
      ZP.PSTRT1 U7 D100 M103  ; 서보 모터 / ZP PD / 기동 성공
61    LD      M103  ; 기동 성공
      ANI     M104  ; 기동 실패
      OR      M601  ; 흡착+
      AND     T600  ; 창고 이동
      OUT     M601  ; 흡착+
66    LD      X0B  ; 흡착 전진
      OR      M602  ; 창고 집기
      AND     M601  ; 흡착+
      OUT     M602  ; 창고 집기
      DECP    D600
